Fanuc KAREL source: kt00192.KL

-- PROVISIONAL review KL for V940-1; original PC SHA256 2a49d92480ee503a171e9ec9f2cb6930885766baf522b2fb28841271a08640c3
-- Incomplete behavior may be omitted. Consult companion uncertainty JSON. Do not deploy.
PROGRAM KT00192
%NOLOCKGROUP
VAR
  OUT : REAL
-- UNRESOLVED_DECL H1 type=002017
-- UNRESOLVED_DECL H2 type=002017
BEGIN
  -- V9_ZERO_TABLE_METADATA_HINT layout=0001; no indexed target words; source/name/runtime held
  -- UNRESOLVED_PC offsets 5-19; opcodes 2E,22,9D,33,B4
  -- UNRESOLVED_PC offsets 24-38; opcodes 2E,22,9D,33,B4
  -- UNRESOLVED_PC offsets 43-57; opcodes 2E,22,9D,33,B4
  -- UNRESOLVED_PC offsets 62-76; opcodes 2E,22,9D,33,B4
  -- UNRESOLVED_PC offsets 81-107; opcodes 22,9D,33,B3,22,9D,33,B3,56,64,23
  -- UNRESOLVED_PC offsets 112-116; opcodes 7F
END KT00192
